// SIMATIC STEP 7 (V5.x) project Desbobinador y cizallado
// CPU: CPU 312
// station: Hardware
// station: SIMATIC 300(1)
// station: P_ADR_BUS

SYMBOL_TABLE
"CONTADOR"	C 1	COUNTER	// Cuenta el numero de planchas cortadas
"Global"	DB 1	DB 1
"Modo1"	DB 2	DB 2
"Modo2"	DB 3	DB 3
"INFO_BOB"	DB 4	DB 4
"DESBOBINADO"	FB 1	FB 1	// Función que se encarga del desbobinado
"CIZALLADO"	FB 2	FB 2	// Funcion que se encaga del cizallado de planchas
"MULT_DESBOB"	FB 3	FB 3
"MULT_CIZA"	FB 4	FB 4
"MULT_GEN"	FB 5	FB 5
"CORTAR"	FC 1	FC 1	// Funcion de cortar las planchas
"PESAJE"	FC 2	FC 2	// Función de pesaje
"MODOS"	FC 3	FC 3	// Gestión de modos
"SCALE"	FC 105	FC 105	// Scaling Values
"PRESENCIA"	I 124.0	BOOL	// Sensor que indica si la bobina está siendo correctamente desbobinada
"SENSOR SARTEN"	I 124.1	BOOL	// Sensor que indica que la plancha ha llegado a la longitud de corte adecuada
"SENSOR CACEROLA"	I 124.2	BOOL	// Sensor que indica que la plancha ha llegado a la longitud de corte adecuada
"SENSOR WOK"	I 124.3	BOOL	// Sensor que indica que la plancha ha llegado a la longitud de corte adecuada
"SENSOR PAELLERA"	I 124.4	BOOL	// Sensor que indica que la plancha ha llegado a la longitud de corte adecuada
"BOBINA COLOCADA"	I 124.5	BOOL	// Sensor que detecta si una bobina ha sido puesta en su lugar para empezar proceso
"SENSOR ABAJO"	I 124.6	BOOL	// Sensor que detecta que la cuchilla de cizallado está abajo
"SENSOR ARRIBA"	I 124.7	BOOL	// Sensor que detecta que la cuchilla de cizallado está arriba
"EXPULSADA"	I 125.0	BOOL	// Sensor que detecta que la plancha recien cortada es expulsada
"MODO A"	I 125.1	BOOL	// Funcionamiento en modo A
"MODO B"	I 125.2	BOOL	// Funcionamiento en modo B
"PALET"	I 125.3	BOOL
"PON"	I 125.4	BOOL
"POFF"	I 125.5	BOOL
"BIT_DE_TRABAJO"	I 125.6	BOOL
"SARTEN"	M 100.1	BOOL	// Peso que corresponde a la bobina para hacer sartenes
"CACEROLA"	M 100.2	BOOL	// Peso que corresponde a la bobina para hacer cacerolas
"WOK"	M 100.3	BOOL	// Peso que corresponde a la bobina para hacer woks
"PAELLERA"	M 100.4	BOOL	// Peso que corresponde a la bobina para hacer paelleras
"CORTADO"	M 100.5	BOOL	// Indica que una plancha ha sido cortada
"X0"	M 101.0	BOOL
"X1"	M 101.1	BOOL
"X2"	M 101.2	BOOL
"X3"	M 101.3	BOOL
"X4"	M 101.4	BOOL
"X5"	M 101.5	BOOL
"X6"	M 101.6	BOOL
"X7"	M 101.7	BOOL
"X8"	M 102.0	BOOL
"X10"	M 102.2	BOOL
"X11"	M 102.3	BOOL
"X20"	M 103.4	BOOL
"X21"	M 103.5	BOOL
"X22"	M 103.6	BOOL
"X23"	M 103.7	BOOL
"X24"	M 104.0	BOOL
"X25"	M 104.1	BOOL
"X30"	M 104.2	BOOL
"X60"	M 104.3	BOOL
"X61"	M 104.4	BOOL
"X62"	M 104.5	BOOL
"X31"	M 104.6	BOOL
"X32"	M 104.7	BOOL
"X33"	M 105.0	BOOL
"X34"	M 105.1	BOOL
"X35"	M 105.2	BOOL
"X40"	M 105.7	BOOL
"X41"	M 106.0	BOOL
"X42"	M 106.1	BOOL
"X43"	M 106.2	BOOL
"X44"	M 106.3	BOOL
"X50"	M 106.7	BOOL
"X51"	M 107.0	BOOL
"X52"	M 107.1	BOOL
"X100"	M 107.2	BOOL
"X101"	M 107.3	BOOL
"X110"	M 107.4	BOOL
"X111"	M 107.5	BOOL
"X53"	M 107.6	BOOL
"X120"	M 107.7	BOOL
"ENDCOUNT"	M 108.0	BOOL	// Marca que avisa del final de la cuenta
"X123"	M 108.2	BOOL
"X124"	M 108.3	BOOL
"X122"	M 108.4	BOOL
"X121"	M 108.5	BOOL
"X54"	M 108.6	BOOL
"STBYDESBOB"	M 108.7	BOOL	// Indica el estado stby del FB1 (desbobinado)
"INIDESBOB"	M 109.0	BOOL	// FP para iniciar el FB1
"INICIZA"	M 109.1	BOOL	// FP para iniciar el FB2
"PLANCHAS"	MW 3	INT	// Numero de planchas por bobina
"OB1"	OB 1	OB 1	// Main programa
"OB100"	OB 100	OB 100	// Inicio del programa
"PESO"	PIW 751	INT	// Sensor de peso que pesa las bobinas
"CENTRO"	PIW 761	INT	// Medida actual del centro
"C_CACEROLA"	PIW 771	INT
"C_SARTEN"	PIW 773	INT
"C_WOK"	PIW 775	INT
"C_PAELLERA"	PIW 777	INT
"ABRIR MCENTRO"	Q 124.1	BOOL	// Salida que hace más grande el centro de sujeción de la bobina
"CERRAR MCENTRO"	Q 124.2	BOOL	// Salida que hace más pequeño el centro de sujeción de la bobina
"DESBOBINAR"	Q 124.3	BOOL	// Actuador que activa la rotación del centro
"EXPULSAR BOBINA"	Q 124.4	BOOL	// Actuador que expulsa el centro de la bobina una vez ha acabado de desbobinar
"BAJAR CUCHILLA"	Q 124.5	BOOL	// Baja la cuchilla, si está a 0 la cuchilla sube
"EXPULSAR PALET"	Q 124.6	BOOL	// Activa un piston que expulsa la plancgha de la zona de corte
"PRENSA"	Q 124.7	BOOL	// Activa la prensa
END_SYMBOL_TABLE

FUNCTION_BLOCK "DESBOBINADO"	// FB 1
TITLE = DESBOBINADO
VERSION : 0.1
VAR_INPUT
  SENSOR : BOOL ;
  PRESENCIA : BOOL ;
  CENTRO : INT ;
  bit_de_trabajo : BOOL ;
  MCENTRO : INT ;
  Contador : COUNTER ;
  START : BOOL ;
  PLANCHAS : WORD  := W#16#100;
END_VAR
VAR_OUTPUT
  ABRIRMCENTRO : BOOL ;
  DESBOBINAR : BOOL ;
  STBY : BOOL ;
END_VAR
VAR
  x31 : BOOL ;
  x32 : BOOL ;
  x33 : BOOL ;
  x34 : BOOL ;
  s1 : BOOL ;
  FP_Bit_Tr : BOOL ;
  x30 : BOOL ;
  FP_PRESENCIA : BOOL ;
  FP_BDT : BOOL ;
  FP_START : BOOL ;
END_VAR
VAR_TEMP
  watchdog_master : BOOL ;
END_VAR
BEGIN
NETWORK
TITLE = Arranque
      SET;
      A     #bit_de_trabajo;
      FP    #FP_BDT;
      S     #x30;
      R     #x31;
      R     #x32;
      R     #x33;
      R     #x34;
      R     #s1;
NETWORK
TITLE = x31 a x32
//Comparacion medida centro con medida nominal del centro para pasar de x31 a x32
      A     #x31;
      A(;
      L     #CENTRO;
      L     #MCENTRO;
      ==R;
      );
      R     #x31;
      S     #x32;
NETWORK
TITLE = x32 a x33
//Presencia detecta que la plancha esta en posicion para empezar el proceso de 
//desbobinado-cizallado
      A     #x32;
      A     #PRESENCIA;
      FP    #FP_PRESENCIA;
      R     #x32;
      S     #x33;
NETWORK
TITLE = x33 a x34
//Detecta que la plancha esta lista para ser cizallada
      A     #x33;
      A     #SENSOR;
      R     #x33;
      S     #x34;
NETWORK
TITLE = x34 a x33
//si el contador no ha acabado
      A     #x34;
      T     LD 1;
      TAK;
      T     LD 5;
      L     #Contador;
      T     LW 9;
      L     LD 5;
      L     LD 1;
      A     C [LW 9];
      AN    #SENSOR;
      R     #x34;
      S     #x33;
NETWORK
TITLE = x34 a s1
//si el contador ha cabado
      A     #x34;
      T     LD 1;
      TAK;
      T     LD 5;
      L     #Contador;
      T     LW 9;
      L     LD 5;
      L     LD 1;
      AN    C [LW 9];
      AN    #SENSOR;
      AN    #PRESENCIA;
      R     #x34;
      S     #x30;
NETWORK
TITLE = Tratamiento de bit de fin
      A     #x30;
      =     #STBY;
NETWORK
TITLE = Abrir centro
      A     #x31;
      =     #ABRIRMCENTRO;
NETWORK
TITLE = Carga del contador y desbobinado en x32
      A     #x32;
      S     #DESBOBINAR;
      L     #PLANCHAS;
      T     LD 1;
      TAK;
      T     LD 5;
      L     #Contador;
      T     LW 9;
      L     LD 5;
      L     LD 1;
      S     C [LW 9];
NETWORK
TITLE = Resta del contador y salida del x33
      A     #x33;
      S     #DESBOBINAR;
NETWORK
TITLE =
      A     #x34;
      R     #DESBOBINAR;
NETWORK
TITLE = De X30 a X31
      A     #x30;
      A     #START;
      FP    #FP_START;
      R     #x30;
      S     #x31;
END_FUNCTION_BLOCK

FUNCTION_BLOCK "CIZALLADO"	// FB 2
TITLE = CIZALLADO
VERSION : 0.1
VAR_INPUT
  bit_de_trabajo : BOOL ;
  SENSOR : BOOL ;
  PLANCHAS : INT ;
  SENSORABAJO : BOOL ;
  SENSORARRIBA : BOOL ;
  EXPULSADA : BOOL ;
  CONTADOR : COUNTER ;
  START : BOOL ;
  STOP : BOOL ;
END_VAR
VAR_OUTPUT
  BAJARCUCHILLA : BOOL ;
  EXPULSARPLANCHA : BOOL ;
  bit_ok : BOOL ;
  bit_error : BOOL ;
  STBY : BOOL ;
END_VAR
VAR
  INICORTAR : BOOL ;
  CORTADO : BOOL ;
  X41 : BOOL ;
  M3 : BOOL ;
  X43 : BOOL ;
  S2 : BOOL ;
  MARCHA : BOOL ;
  PARO : BOOL ;
END_VAR
BEGIN
NETWORK
TITLE = Arranque
      SET;
      FP    #bit_de_trabajo;
      S     #X41;
      R     #M3;
      R     #X43;
      R     #INICORTAR;
      R     #CORTADO;
      R     #bit_ok;
      R     #bit_error;
      R     #S2;
NETWORK
TITLE = De x41 a M3
      A     #X41;
      A     #SENSOR;
      A     #MARCHA;
      R     #X41;
      S     #M3;
NETWORK
TITLE = De M3 a x43
      A     #M3;
      A     #CORTADO;
      R     #M3;
      S     #X43;
NETWORK
TITLE = de x43 a x41
      A     #X43;
      T     LD 0;
      TAK;
      T     LD 4;
      L     #CONTADOR;
      T     LW 8;
      L     LD 4;
      L     LD 0;
      AN    C [LW 8];
      R     #X43;
      S     #X41;
NETWORK
TITLE = de x43 a s2
      A     #X43;
      T     LD 0;
      TAK;
      T     LD 4;
      L     #CONTADOR;
      T     LW 8;
      L     LD 4;
      L     LD 0;
      A     C [LW 8];
      R     #X43;
      S     #S2;
NETWORK
TITLE = De M3 a x43 con call M3
      A     #M3;
      JCN   _001;
      CALL  "CORTAR" (
           bit_de_trabajo           := #INICORTAR,
           SENSORABAJO              := #SENSORABAJO,
           SENSORARRIBA             := #SENSORARRIBA,
           EXPULSADA                := #EXPULSADA,
           BAJARCUCHILLA            := #BAJARCUCHILLA,
           EXPULSARPLANCHA          := #EXPULSARPLANCHA,
           bit_ok                   := #CORTADO);
_001: NOP   0;
      A     #CORTADO;
      R     #M3;
      S     #X43;
NETWORK
TITLE =
      A     #M3;
      =     #INICORTAR;
NETWORK
TITLE = Cuenta el numero de planchas cortadas
      A     #X43;
      T     LD 0;
      TAK;
      T     LD 4;
      L     #CONTADOR;
      T     LW 8;
      L     LD 4;
      L     LD 0;
      CU    C [LW 8];
NETWORK
TITLE =
      A     #MARCHA;
      A     #STOP;
      R     #MARCHA;
      S     #PARO;
NETWORK
TITLE =
      A     #PARO;
      A     #START;
      AN    #STOP;
      R     #PARO;
      S     #MARCHA;
NETWORK
TITLE =
      A     #S2;
      =     #bit_ok;
END_FUNCTION_BLOCK

FUNCTION_BLOCK "MULT_DESBOB"	// FB 3
VERSION : 0.1
VAR_INPUT
  S_CACEROLA : BOOL ;
  S_SARTEN : BOOL ;
  S_WOK : BOOL ;
  S_PAELLERA : BOOL ;
  PRESENCIA : BOOL ;
  C_CACEROLA : INT ;
  C_SARTEN : INT ;
  C_WOK : INT ;
  C_PAELLERA : INT ;
  BIT_DE_TRABAJO : BOOL ;
  MCENTRO : INT ;
  CONTADOR : COUNTER ;
  START : BOOL ;
  STOP : BOOL ;
  PLANCHAS : WORD ;
  SARTEN : BOOL ;
  CACEROLA : BOOL ;
  WOK : BOOL ;
  PAELLERA : BOOL ;
END_VAR
VAR_OUTPUT
  ABRIRMCENTRO : BOOL ;
  DESBOBINAR : BOOL ;
  BIT_OK : BOOL ;
  BIT_ERROR : BOOL ;
  STBY : BOOL ;
END_VAR
VAR
  CAC_DESB : FB 1;
  SART_DESB : FB 1;
  WOK_DESB : FB 1;
  PAELL_DESB : FB 1;
END_VAR
BEGIN
NETWORK
TITLE =
      A     #SARTEN;
      BLD   14;
      =     L 6.0;
      L     DINO;
      T     LW 4;
      CDB;
      OPN   DI [LW 4];
      TAR2  LD 0;
      A     DBX [AR2,P#0.1];
      =     #SART_DESB.SENSOR;
      A     DBX [AR2,P#0.4];
      =     #SART_DESB.PRESENCIA;
      L     DBW [AR2,P#4.0];
      T     #SART_DESB.CENTRO;
      A     DBX [AR2,P#10.0];
      =     #SART_DESB.bit_de_trabajo;
      L     DBW [AR2,P#12.0];
      T     #SART_DESB.MCENTRO;
      L     DBW [AR2,P#14.0];
      T     #SART_DESB.Contador;
      A     DBX [AR2,P#16.0];
      =     #SART_DESB.START;
      A     DBX [AR2,P#16.1];
      =     DIX [AR2,P#52.1];
      L     DBW [AR2,P#18.0];
      T     #SART_DESB.PLANCHAS;
      +AR2  P#42.0;
      UC    "DESBOBINADO";
      LAR2  LD 0;
      A     #SART_DESB.ABRIRMCENTRO;
      =     DBX [AR2,P#22.0];
      A     #SART_DESB.DESBOBINAR;
      =     DBX [AR2,P#22.1];
      A     #SART_DESB.STBY;
      =     DBX [AR2,P#22.2];
      A     DIX [AR2,P#56.3];
      =     DBX [AR2,P#22.3];
      A     DIX [AR2,P#56.4];
      =     DBX [AR2,P#22.4];
      CDB;
      BLD   15;
NETWORK
TITLE =
      A     #CACEROLA;
      BLD   14;
      =     L 6.0;
      L     DINO;
      T     LW 4;
      CDB;
      OPN   DI [LW 4];
      TAR2  LD 0;
      A     DBX [AR2,P#0.0];
      =     #CAC_DESB.SENSOR;
      A     DBX [AR2,P#0.4];
      =     #CAC_DESB.PRESENCIA;
      L     DBW [AR2,P#2.0];
      T     #CAC_DESB.CENTRO;
      A     DBX [AR2,P#10.0];
      =     #CAC_DESB.bit_de_trabajo;
      L     DBW [AR2,P#12.0];
      T     #CAC_DESB.MCENTRO;
      L     DBW [AR2,P#14.0];
      T     #CAC_DESB.Contador;
      A     DBX [AR2,P#16.0];
      =     #CAC_DESB.START;
      A     DBX [AR2,P#16.1];
      =     DIX [AR2,P#34.1];
      L     DBW [AR2,P#18.0];
      T     #CAC_DESB.PLANCHAS;
      +AR2  P#24.0;
      UC    "DESBOBINADO";
      LAR2  LD 0;
      A     #CAC_DESB.ABRIRMCENTRO;
      =     DBX [AR2,P#22.0];
      A     #CAC_DESB.DESBOBINAR;
      =     DBX [AR2,P#22.1];
      A     #CAC_DESB.STBY;
      =     DBX [AR2,P#22.2];
      A     DIX [AR2,P#38.3];
      =     DBX [AR2,P#22.3];
      A     DIX [AR2,P#38.4];
      =     DBX [AR2,P#22.4];
      CDB;
      BLD   15;
NETWORK
TITLE =
      A     #WOK;
      BLD   14;
      =     L 6.0;
      L     DINO;
      T     LW 4;
      CDB;
      OPN   DI [LW 4];
      TAR2  LD 0;
      A     DBX [AR2,P#0.2];
      =     #WOK_DESB.SENSOR;
      A     DBX [AR2,P#0.4];
      =     #WOK_DESB.PRESENCIA;
      L     DBW [AR2,P#6.0];
      T     #WOK_DESB.CENTRO;
      A     DBX [AR2,P#10.0];
      =     #WOK_DESB.bit_de_trabajo;
      L     DBW [AR2,P#12.0];
      T     #WOK_DESB.MCENTRO;
      L     DBW [AR2,P#14.0];
      T     #WOK_DESB.Contador;
      A     DBX [AR2,P#16.0];
      =     #WOK_DESB.START;
      A     DBX [AR2,P#16.1];
      =     DIX [AR2,P#70.1];
      L     DBW [AR2,P#18.0];
      T     #WOK_DESB.PLANCHAS;
      +AR2  P#60.0;
      UC    "DESBOBINADO";
      LAR2  LD 0;
      A     #WOK_DESB.ABRIRMCENTRO;
      =     DBX [AR2,P#22.0];
      A     #WOK_DESB.DESBOBINAR;
      =     DBX [AR2,P#22.1];
      A     #WOK_DESB.STBY;
      =     DBX [AR2,P#22.2];
      A     DIX [AR2,P#74.3];
      =     DBX [AR2,P#22.3];
      A     DIX [AR2,P#74.4];
      =     DBX [AR2,P#22.4];
      CDB;
      BLD   15;
NETWORK
TITLE =
      A     #PAELLERA;
      BLD   14;
      =     L 6.0;
      L     DINO;
      T     LW 4;
      CDB;
      OPN   DI [LW 4];
      TAR2  LD 0;
      A     DBX [AR2,P#0.3];
      =     #PAELL_DESB.SENSOR;
      A     DBX [AR2,P#0.4];
      =     #PAELL_DESB.PRESENCIA;
      L     DBW [AR2,P#8.0];
      T     #PAELL_DESB.CENTRO;
      A     DBX [AR2,P#10.0];
      =     #PAELL_DESB.bit_de_trabajo;
      L     DBW [AR2,P#12.0];
      T     #PAELL_DESB.MCENTRO;
      L     DBW [AR2,P#14.0];
      T     #PAELL_DESB.Contador;
      A     DBX [AR2,P#16.0];
      =     #PAELL_DESB.START;
      A     DBX [AR2,P#16.1];
      =     DIX [AR2,P#88.1];
      L     DBW [AR2,P#18.0];
      T     #PAELL_DESB.PLANCHAS;
      +AR2  P#78.0;
      UC    "DESBOBINADO";
      LAR2  LD 0;
      A     #PAELL_DESB.ABRIRMCENTRO;
      =     DBX [AR2,P#22.0];
      A     #PAELL_DESB.DESBOBINAR;
      =     DBX [AR2,P#22.1];
      A     #PAELL_DESB.STBY;
      =     DBX [AR2,P#22.2];
      A     DIX [AR2,P#92.3];
      =     DBX [AR2,P#22.3];
      A     DIX [AR2,P#92.4];
      =     DBX [AR2,P#22.4];
      CDB;
      BLD   15;
END_FUNCTION_BLOCK

FUNCTION_BLOCK "MULT_CIZA"	// FB 4
VERSION : 0.1
VAR_INPUT
  S_CACEROLA : BOOL ;
  S_WOK : BOOL ;
  S_SARTEN : BOOL ;
  S_PAELLERA : BOOL ;
  BIT_DE_TRABAJO : BOOL ;
  PLANCHAS : INT ;
  SENSORARRIBA : BOOL ;
  SENSORABAJO : BOOL ;
  EXPULSADA : BOOL ;
  CONTADOR : COUNTER ;
  SARTEN : BOOL ;
  CACEROLA : BOOL ;
  WOK : BOOL ;
  PAELLERA : BOOL ;
  START : BOOL ;
  STOP : BOOL ;
END_VAR
VAR_OUTPUT
  EXPULSARPLANCHA : BOOL ;
  BAJARCUCHILLA : BOOL ;
  BIT_OK : BOOL ;
END_VAR
VAR
  CAC_CIZA : FB 2;
  SART_CIZA : FB 2;
  WOK_CIZA : FB 2;
  PAELL_CIZA : FB 2;
  STBY : BOOL ;
END_VAR
BEGIN
NETWORK
TITLE =
      A     #CACEROLA;
      BLD   14;
      =     L 6.0;
      L     DINO;
      T     LW 4;
      CDB;
      OPN   DI [LW 4];
      TAR2  LD 0;
      A     DBX [AR2,P#0.4];
      =     #CAC_CIZA.bit_de_trabajo;
      A     DBX [AR2,P#0.0];
      =     #CAC_CIZA.SENSOR;
      L     DBW [AR2,P#2.0];
      T     #CAC_CIZA.PLANCHAS;
      A     DBX [AR2,P#4.1];
      =     #CAC_CIZA.SENSORABAJO;
      A     DBX [AR2,P#4.0];
      =     #CAC_CIZA.SENSORARRIBA;
      A     DBX [AR2,P#4.2];
      =     #CAC_CIZA.EXPULSADA;
      L     DBW [AR2,P#6.0];
      T     #CAC_CIZA.CONTADOR;
      A     DBX [AR2,P#8.4];
      =     #CAC_CIZA.START;
      A     DBX [AR2,P#8.5];
      =     #CAC_CIZA.STOP;
      +AR2  P#12.0;
      UC    "CIZALLADO";
      LAR2  LD 0;
      A     #CAC_CIZA.BAJARCUCHILLA;
      =     DBX [AR2,P#10.1];
      A     #CAC_CIZA.EXPULSARPLANCHA;
      =     DBX [AR2,P#10.0];
      A     #CAC_CIZA.bit_ok;
      =     DBX [AR2,P#10.2];
      A     #CAC_CIZA.STBY;
      =     DBX [AR2,P#68.0];
      CDB;
      BLD   15;
NETWORK
TITLE =
      A     #WOK;
      BLD   14;
      =     L 6.0;
      L     DINO;
      T     LW 4;
      CDB;
      OPN   DI [LW 4];
      TAR2  LD 0;
      A     DBX [AR2,P#0.4];
      =     #WOK_CIZA.bit_de_trabajo;
      A     DBX [AR2,P#0.1];
      =     #WOK_CIZA.SENSOR;
      L     DBW [AR2,P#2.0];
      T     #WOK_CIZA.PLANCHAS;
      A     DBX [AR2,P#4.1];
      =     #WOK_CIZA.SENSORABAJO;
      A     DBX [AR2,P#4.0];
      =     #WOK_CIZA.SENSORARRIBA;
      A     DBX [AR2,P#4.2];
      =     #WOK_CIZA.EXPULSADA;
      L     DBW [AR2,P#6.0];
      T     #WOK_CIZA.CONTADOR;
      A     DBX [AR2,P#8.4];
      =     #WOK_CIZA.START;
      A     DBX [AR2,P#8.5];
      =     #WOK_CIZA.STOP;
      +AR2  P#40.0;
      UC    "CIZALLADO";
      LAR2  LD 0;
      A     #WOK_CIZA.BAJARCUCHILLA;
      =     DBX [AR2,P#10.1];
      A     #WOK_CIZA.EXPULSARPLANCHA;
      =     DBX [AR2,P#10.0];
      A     #WOK_CIZA.bit_ok;
      =     DBX [AR2,P#10.2];
      A     #WOK_CIZA.STBY;
      =     DBX [AR2,P#68.0];
      CDB;
      BLD   15;
NETWORK
TITLE =
      A     #SARTEN;
      BLD   14;
      =     L 6.0;
      L     DINO;
      T     LW 4;
      CDB;
      OPN   DI [LW 4];
      TAR2  LD 0;
      A     DBX [AR2,P#0.4];
      =     #SART_CIZA.bit_de_trabajo;
      A     DBX [AR2,P#0.2];
      =     #SART_CIZA.SENSOR;
      L     DBW [AR2,P#2.0];
      T     #SART_CIZA.PLANCHAS;
      A     DBX [AR2,P#4.1];
      =     #SART_CIZA.SENSORABAJO;
      A     DBX [AR2,P#4.0];
      =     #SART_CIZA.SENSORARRIBA;
      A     DBX [AR2,P#4.2];
      =     #SART_CIZA.EXPULSADA;
      L     DBW [AR2,P#6.0];
      T     #SART_CIZA.CONTADOR;
      A     DBX [AR2,P#8.4];
      =     #SART_CIZA.START;
      A     DBX [AR2,P#8.5];
      =     #SART_CIZA.STOP;
      +AR2  P#26.0;
      UC    "CIZALLADO";
      LAR2  LD 0;
      A     #SART_CIZA.BAJARCUCHILLA;
      =     DBX [AR2,P#10.1];
      A     #SART_CIZA.EXPULSARPLANCHA;
      =     DBX [AR2,P#10.0];
      A     #SART_CIZA.bit_ok;
      =     DBX [AR2,P#10.2];
      A     #SART_CIZA.STBY;
      =     DBX [AR2,P#68.0];
      CDB;
      BLD   15;
NETWORK
TITLE =
      A     #PAELLERA;
      BLD   14;
      =     L 6.0;
      L     DINO;
      T     LW 4;
      CDB;
      OPN   DI [LW 4];
      TAR2  LD 0;
      A     DBX [AR2,P#0.4];
      =     #PAELL_CIZA.bit_de_trabajo;
      A     DBX [AR2,P#0.3];
      =     #PAELL_CIZA.SENSOR;
      L     DBW [AR2,P#2.0];
      T     #PAELL_CIZA.PLANCHAS;
      A     DBX [AR2,P#4.1];
      =     #PAELL_CIZA.SENSORABAJO;
      A     DBX [AR2,P#4.0];
      =     #PAELL_CIZA.SENSORARRIBA;
      A     DBX [AR2,P#4.2];
      =     #PAELL_CIZA.EXPULSADA;
      L     DBW [AR2,P#6.0];
      T     #PAELL_CIZA.CONTADOR;
      A     DBX [AR2,P#8.4];
      =     #PAELL_CIZA.START;
      A     DBX [AR2,P#8.5];
      =     #PAELL_CIZA.STOP;
      +AR2  P#54.0;
      UC    "CIZALLADO";
      LAR2  LD 0;
      A     #PAELL_CIZA.BAJARCUCHILLA;
      =     DBX [AR2,P#10.1];
      A     #PAELL_CIZA.EXPULSARPLANCHA;
      =     DBX [AR2,P#10.0];
      A     #PAELL_CIZA.bit_ok;
      =     DBX [AR2,P#10.2];
      A     #PAELL_CIZA.STBY;
      =     DBX [AR2,P#68.0];
      CDB;
      BLD   15;
END_FUNCTION_BLOCK

FUNCTION_BLOCK "MULT_GEN"	// FB 5
VERSION : 0.1
VAR_INPUT
  MODO : BOOL ;
  BIT_DE_TRABAJO : BOOL ;
  START : BOOL ;
  STOP : BOOL ;
  BOBINA_COLOCADA : BOOL ;
  IN_SCALE : INT ;
  S_CACEROLA : BOOL ;
  S_WOK : BOOL ;
  S_PAELLERA : BOOL ;
  S_SARTEN : BOOL ;
  PRESENCIA : BOOL ;
  MCENTRO : INT ;
  CONTADOR : COUNTER ;
END_VAR
VAR_OUTPUT
  ABRIRMCENTRO : BOOL ;
END_VAR
VAR_IN_OUT
  DESBOBINAR : BOOL ;
END_VAR
VAR
  CIZALLADO : FB 4;
  DESBOBINADO : FB 3;
  X0 : BOOL ;
  MARCHA : BOOL ;
  PARO : BOOL ;
  X1 : BOOL ;
  M4 : BOOL ;
  M1 : BOOL ;
  X7 : BOOL ;
  X8 : BOOL ;
  X10 : BOOL ;
  X11 : BOOL ;
  X20 : BOOL ;
  M2 : BOOL ;
  X25 : BOOL ;
  OK_SCALE : BOOL ;
  START_SCALE : BOOL ;
  STOP_SCALE : BOOL ;
  STBY_SCALE : BOOL ;
  SARTEN : BOOL ;
  CACEROLA : BOOL ;
  WOK : BOOL ;
  PAELLERA : BOOL ;
  START_DESBOBINADO : BOOL ;
  STOP_DESBOBINADO : BOOL ;
END_VAR
BEGIN
NETWORK
TITLE =
      A     #BIT_DE_TRABAJO;
      S     #X0;
      S     #PARO;
      R     #MARCHA;
      R     #X1;
      R     #M4;
      R     #M1;
      R     #X7;
      R     #X8;
      R     #X10;
      R     #X11;
      R     #X20;
      R     #M2;
      R     #X25;
NETWORK
TITLE =
      A     #MARCHA;
      A     #STOP;
      R     #MARCHA;
      S     #PARO;
NETWORK
TITLE =
      A     #PARO;
      A     #START;
      AN    #STOP;
      R     #PARO;
      S     #MARCHA;
NETWORK
TITLE =
      A     #X0;
      A     #MARCHA;
      R     #X0;
      S     #X1;
      S     #X10;
      S     #X20;
NETWORK
TITLE =
      A     #X1;
      A     #BOBINA_COLOCADA;
      R     #X1;
      S     #M4;
NETWORK
TITLE =
      A     #M4;
      JCN   _001;
      CALL  "PESAJE" (
           in                       := #IN_SCALE,
           PESO_SARTEN              := "Global".PESO_SARTEN,
           PESO_CACEROLA            := "Global".PESO_CACEROLA,
           PESO_WOK                 := "Global".PESO_WOK,
           PESO_PAELLERA            := "Global".PESO_PAELLERA,
           bit_de_trabajo           := #BIT_DE_TRABAJO,
           RECIBIDO                 := #OK_SCALE,
           START                    := #START_SCALE,
           STOP                     := #STOP_SCALE,
           stby                     := #STBY_SCALE,
           SARTEN                   := #SARTEN,
           CACEROLA                 := #CACEROLA,
           WOK                      := #WOK,
           PAELLERA                 := #PAELLERA);
_001: NOP   0;
NETWORK
TITLE =
      A     #M4;
      =     #START_SCALE;
NETWORK
TITLE =
      A     #M4;
      A(;
      A     #SARTEN;
      O     #WOK;
      O     #PAELLERA;
      O     #CACEROLA;
      );
      JCN   _002;
      BLD   14;
      =     L 6.0;
      L     DINO;
      T     LW 4;
      CDB;
      OPN   DI [LW 4];
      TAR2  LD 0;
      A     DBX [AR2,P#4.0];
      =     #DESBOBINADO.S_CACEROLA;
      A     DBX [AR2,P#4.3];
      =     #DESBOBINADO.S_SARTEN;
      A     DBX [AR2,P#4.1];
      =     #DESBOBINADO.S_WOK;
      A     DBX [AR2,P#4.2];
      =     #DESBOBINADO.S_PAELLERA;
      A     DBX [AR2,P#4.4];
      =     #DESBOBINADO.PRESENCIA;
      OPN   DI 4;
      L     DIW 0;
      OPN   DI [LW 4];
      T     #DESBOBINADO.C_CACEROLA;
      OPN   DI 4;
      L     DIW 2;
      OPN   DI [LW 4];
      T     #DESBOBINADO.C_SARTEN;
      OPN   DI 4;
      L     DIW 4;
      OPN   DI [LW 4];
      T     #DESBOBINADO.C_WOK;
      OPN   DI 4;
      L     DIW 6;
      OPN   DI [LW 4];
      T     #DESBOBINADO.C_PAELLERA;
      A     DBX [AR2,P#0.1];
      =     #DESBOBINADO.BIT_DE_TRABAJO;
      L     DBW [AR2,P#6.0];
      T     #DESBOBINADO.MCENTRO;
      L     DBW [AR2,P#8.0];
      T     #DESBOBINADO.CONTADOR;
      A     DBX [AR2,P#182.5];
      =     #DESBOBINADO.START;
      A     DBX [AR2,P#182.6];
      =     #DESBOBINADO.STOP;
      OPN   DI 1;
      L     DIW 16;
      OPN   DI [LW 4];
      T     #DESBOBINADO.PLANCHAS;
      A     DBX [AR2,P#182.1];
      =     #DESBOBINADO.SARTEN;
      A     DBX [AR2,P#182.2];
      =     #DESBOBINADO.CACEROLA;
      A     DBX [AR2,P#182.3];
      =     #DESBOBINADO.WOK;
      A     DBX [AR2,P#182.4];
      =     #DESBOBINADO.PAELLERA;
      +AR2  P#84.0;
      UC    "MULT_DESBOB";
      LAR2  LD 0;
      A     #DESBOBINADO.ABRIRMCENTRO;
      =     DBX [AR2,P#10.0];
      A     #DESBOBINADO.DESBOBINAR;
      =     DBX [AR2,P#12.0];
      CDB;
      BLD   15;
_002: NOP   0;
END_FUNCTION_BLOCK

FUNCTION "CORTAR" : VOID	// FC 1
TITLE = CORTAR
VERSION : 0.1
VAR_INPUT
  bit_de_trabajo : BOOL ;
  SENSORABAJO : BOOL ;
  SENSORARRIBA : BOOL ;
  EXPULSADA : BOOL ;
END_VAR
VAR_OUTPUT
  BAJARCUCHILLA : BOOL ;
  EXPULSARPLANCHA : BOOL ;
  bit_ok : BOOL ;
END_VAR
VAR_TEMP
  x51 : BOOL ;
  x52 : BOOL ;
  x53 : BOOL ;
  s3 : BOOL ;
END_VAR
BEGIN
NETWORK
TITLE = Arranque
      SET;
      FP    #bit_de_trabajo;
      S     #x51;
      R     #x52;
      R     #x53;
      R     #s3;
NETWORK
TITLE = de x51 a x52
      A     #x51;
      A     #SENSORABAJO;
      R     #x51;
      S     #x52;
NETWORK
TITLE = de x52 a x53
      A     #x52;
      A     #SENSORARRIBA;
      R     #x52;
      S     #x53;
NETWORK
TITLE = de x53 a s3
      A     #x53;
      A     #EXPULSADA;
      R     #x53;
      S     #s3;
NETWORK
TITLE = Accion x51
      A     "X51";
      =     #BAJARCUCHILLA;
NETWORK
TITLE = Accion x53
      A     #x53;
      =     #EXPULSARPLANCHA;
NETWORK
TITLE = Accion final
      A     #s3;
      =     #bit_ok;
END_FUNCTION

FUNCTION "PESAJE" : VOID	// FC 2
TITLE = PESAJE
VERSION : 0.1
VAR_INPUT
  in : INT ;
  PESO_SARTEN : REAL ;
  PESO_CACEROLA : REAL ;
  PESO_WOK : REAL ;
  PESO_PAELLERA : REAL ;
  bit_de_trabajo : BOOL ;
  RECIBIDO : BOOL ;
  START : BOOL ;
  STOP : BOOL ;
END_VAR
VAR_OUTPUT
  stby : BOOL ;
  SARTEN : BOOL ;
  CACEROLA : BOOL ;
  WOK : BOOL ;
  PAELLERA : BOOL ;
END_VAR
VAR_TEMP
  retFC105 : WORD ;
  PESO : REAL ;
  x121 : BOOL ;
  x122 : BOOL ;
  x123 : BOOL ;
  x124 : BOOL ;
  m3 : BOOL ;
  x120 : BOOL ;
  MARCHA : BOOL ;
  PARO : BOOL ;
END_VAR
BEGIN
NETWORK
TITLE = Pesado
      A     #m3;
      CALL  "SCALE" (
           $1                       := #in,
           $2                       := L#1133903872,
           $3                       := L#0,
           $4                       := FALSE,
           $5                       := #retFC105,
           $6                       := #PESO);
NETWORK
TITLE = Arranque
      SET;
      FP    #bit_de_trabajo;
      S     #m3;
      R     #x121;
      R     #x122;
      R     #x123;
      R     #x124;
NETWORK
TITLE = COMPARACION PESO CON PESO_SARTEN
      A(;
      L     #PESO;
      A(;
      L     #PESO_SARTEN;
      L     5.000000e+00;
      +R;
      );
      <=R;
      );
      A(;
      L     #PESO;
      A(;
      L     #PESO_SARTEN;
      L     5.000000e+00;
      -R;
      );
      >=R;
      );
      A     #MARCHA;
      S     #x121;
      R     #m3;
NETWORK
TITLE = COMPARACION PESO CON PESO_CACEROLA
      A(;
      L     #PESO;
      A(;
      L     #PESO_CACEROLA;
      L     5.000000e+00;
      +R;
      );
      <=R;
      );
      A(;
      L     #PESO;
      A(;
      L     #PESO_CACEROLA;
      L     5.000000e+00;
      -R;
      );
      >=R;
      );
      A     #MARCHA;
      S     #x122;
      R     #m3;
NETWORK
TITLE = COMPARACION PESO PESO_WOK
      A(;
      L     #PESO;
      A(;
      L     #PESO_WOK;
      L     5.000000e+00;
      +R;
      );
      <=R;
      );
      A(;
      L     #PESO;
      A(;
      L     #PESO_WOK;
      L     5.000000e+00;
      -R;
      );
      >=R;
      );
      A     #MARCHA;
      S     #x123;
      R     #m3;
NETWORK
TITLE = COMPARACION PESO CON PESO_PAELLERA
      A(;
      L     #PESO;
      A(;
      L     #PESO_PAELLERA;
      L     5.000000e+00;
      +R;
      );
      <=R;
      );
      A(;
      L     #PESO;
      A(;
      L     #PESO_PAELLERA;
      L     5.000000e+00;
      -R;
      );
      >=R;
      );
      A     #MARCHA;
      S     #x124;
      R     #m3;
NETWORK
TITLE = TRATAMIENTO SALIDAS
      A     #x121;
      =     #SARTEN;
      A     #x122;
      =     #CACEROLA;
      A     #x123;
      =     #WOK;
      A     #x124;
      =     #PAELLERA;
NETWORK
TITLE = Paso de estado pesado a stby
      A(;
      A     #x121;
      O     #x122;
      O     #x123;
      O     #x124;
      );
      A     #RECIBIDO;
      R     #x121;
      R     #x122;
      R     #x123;
      R     #x124;
      S     #x120;
NETWORK
TITLE = Salida STBY
      A     #x120;
      =     #stby;
NETWORK
TITLE = MARCHA PARO
      A     #MARCHA;
      A     #STOP;
      R     #MARCHA;
      S     #PARO;
NETWORK
TITLE = PARO MARCHA
      A     #PARO;
      A     #START;
      AN    #STOP;
      R     #PARO;
      S     #MARCHA;
END_FUNCTION

FUNCTION "MODOS" : VOID	// FC 3
TITLE = GESTION DE MODOS
VERSION : 0.1
VAR_INPUT
  MODO1 : BOOL ;
  MODO2 : BOOL ;
END_VAR
VAR_OUTPUT
  CONTADOR : INT ;
  PSARTEN : INT ;
  PCACEROLA : INT ;
  PWOK : INT ;
  PPAELLERA : INT ;
END_VAR
VAR_TEMP
  X60 : BOOL ;
  X61 : BOOL ;
  X62 : BOOL ;
END_VAR
BEGIN
NETWORK
TITLE = De X60 a X61
      A     #X60;
      A     #MODO1;
      R     #X60;
      S     #X61;
NETWORK
TITLE = De X61 a X60
      A     #X61;
      AN    #MODO1;
      R     #X61;
      S     #X60;
NETWORK
TITLE = De X60 a X62
      A     #X60;
      A     #MODO2;
      R     #X60;
      S     #X62;
NETWORK
TITLE = De X62 a X60
      A     #X62;
      AN    #MODO2;
      R     #X62;
      S     #X60;
NETWORK
TITLE = Numero de planchas por bobina y peso Modo 1
      A     #X61;
      L     "Modo1".PLANCHAS;
      T     "Global".PLANCHAS;
      L     "Modo1".PESO_PAELLERA;
      T     "Global".PESO_PAELLERA;
      L     "Modo1".PESO_WOK;
      T     "Global".PESO_WOK;
      L     "Modo1".PESO_SARTEN;
      T     "Global".PESO_SARTEN;
      L     "Modo1".PESO_CACEROLA;
      T     "Global".PESO_CACEROLA;
NETWORK
TITLE =
      A     #X62;
      L     "Modo2".PLANCHAS;
      T     "Global".PLANCHAS;
      L     "Modo2".PESO_PAELLERA;
      T     "Global".PESO_PAELLERA;
      L     "Modo2".PESO_WOK;
      T     "Global".PESO_WOK;
      L     "Modo2".PESO_SARTEN;
      T     "Global".PESO_SARTEN;
      L     "Modo2".PESO_CACEROLA;
      T     "Global".PESO_CACEROLA;
NETWORK
TITLE = Numero de planchas por bobina y peso Modo 2
      A     #X62;
      L     #CONTADOR;
      OPN   DB 200;
      L     #PSARTEN;
      OPN   DB 200;
      L     #PCACEROLA;
      OPN   DB 220;
      L     #PWOK;
      OPN   DB 240;
      L     #PPAELLERA;
      OPN   DB 260;
END_FUNCTION

// FC 105: know-how protected block, not included

DATA_BLOCK "Global"	// DB 1
VERSION : 0.1
  STRUCT
   PESO_CACEROLA : REAL ;	//Peso Bobina Cacerolas
   PESO_WOK : REAL ;	//Peso Bobina Wok
   PESO_SARTEN : REAL ;	//Peso Bobina Sarten
   PESO_PAELLERA : REAL ;	//Peso Bobina Paellera
   PLANCHAS : WORD ;	//Número de planchas por bobina
  END_STRUCT ;	
BEGIN
   PESO_CACEROLA := 1.000000e+02;
   PESO_WOK := 1.100000e+02;
   PESO_SARTEN := 1.200000e+02;
   PESO_PAELLERA := 1.300000e+02;
   PLANCHAS := W#16#100;
END_DATA_BLOCK

DATA_BLOCK "Modo1"	// DB 2
VERSION : 0.1
  STRUCT
   PESO_CACEROLA : REAL  := 1.000000e+002;	//Peso Bobina Cacerolas
   PESO_WOK : REAL  := 1.100000e+002;	//Peso Bobina Wok
   PESO_SARTEN : REAL  := 1.200000e+002;	//Peso Bobina Sarten
   PESO_PAELLERA : REAL  := 1.300000e+002;	//Peso Bobina Paellera
   PLANCHAS : WORD  := W#16#100;	//Número de planchas por bobina
  END_STRUCT ;	
BEGIN
   PESO_CACEROLA := 1.000000e+02;
   PESO_WOK := 1.100000e+02;
   PESO_SARTEN := 1.200000e+02;
   PESO_PAELLERA := 1.300000e+02;
   PLANCHAS := W#16#100;
END_DATA_BLOCK

DATA_BLOCK "Modo2"	// DB 3
VERSION : 0.1
  STRUCT
   PESO_CACEROLA : REAL  := 2.000000e+002;	//Peso Bobina Cacerolas
   PESO_WOK : REAL  := 2.200000e+002;	//Peso Bobina Wok
   PESO_SARTEN : REAL  := 2.400000e+002;	//Peso Bobina Sarten
   PESO_PAELLERA : REAL  := 2.600000e+002;	//Peso Bobina Paellera
   PLANCHAS : WORD  := W#16#200;	//Número de planchas por bobina
  END_STRUCT ;	
BEGIN
   PESO_CACEROLA := 2.000000e+02;
   PESO_WOK := 2.200000e+02;
   PESO_SARTEN := 2.400000e+02;
   PESO_PAELLERA := 2.600000e+02;
   PLANCHAS := W#16#200;
END_DATA_BLOCK

DATA_BLOCK "INFO_BOB"	// DB 4
VERSION : 0.1
  STRUCT
   CENTRO_CACEROLA : INT ;	//Variable provisional
   CENTRO_SARTEN : INT ;
   CENTRO_WOK : INT ;
   CENTRO_PAELLERA : INT ;
  END_STRUCT ;	
BEGIN
END_DATA_BLOCK

ORGANIZATION_BLOCK "OB1"	// OB 1
TITLE = "Main Program Sweep (Cycle)"
VERSION : 0.1
VAR_TEMP
  OB1_EV_CLASS : BYTE ;	//Bits 0-3 = 1 (Coming event), Bits 4-7 = 1 (Event class 1)
  OB1_SCAN_1 : BYTE ;	//1 (Cold restart scan 1 of OB 1), 3 (Scan 2-n of OB 1)
  OB1_PRIORITY : BYTE ;	//Priority of OB Execution
  OB1_OB_NUMBR : BYTE ;	//1 (Organization block 1, OB1)
  OB1_RESERVED_1 : BYTE ;	//Reserved for system
  OB1_RESERVED_2 : BYTE ;	//Reserved for system
  OB1_PREV_CYCLE : INT ;	//Cycle time of previous OB1 scan (milliseconds)
  OB1_MIN_CYCLE : INT ;	//Minimum cycle time of OB1 (milliseconds)
  OB1_MAX_CYCLE : INT ;	//Maximum cycle time of OB1 (milliseconds)
  OB1_DATE_TIME : DATE_AND_TIME ;	//Date and time OB1 started
END_VAR
BEGIN
NETWORK
TITLE =
      A     "X100";
      A     "PON";
      AN    "POFF";
      R     "X100";
      S     "X101";
NETWORK
TITLE =
      A     "X101";
      A     "POFF";
      R     "X101";
      S     "X100";
NETWORK
TITLE =
      A     "X0";
      A     "X101";
      AN    "X60";
      R     "X0";
      S     "X1";
      S     "X10";
      S     "X20";
NETWORK
TITLE =
      A     "X1";
      A     "BOBINA COLOCADA";
      R     "X1";
      S     "X2";
NETWORK
TITLE =
      A     "X2";
      A     DB1.DBX 4.1;
      R     "X2";
      S     "X3";
NETWORK
TITLE =
      A     "X2";
      A     DB2.DBX 4.1;
      R     "X2";
      S     "X4";
NETWORK
TITLE =
      A     "X2";
      A     DB3.DBX 4.1;
      R     "X2";
      S     "X5";
NETWORK
TITLE =
      A     "X2";
      A     DB4.DBX 4.1;
      R     "X2";
      S     "X6";
NETWORK
TITLE =
      A     "X3";
      O     "X4";
      O     "X5";
      O     "X6";
      R     "X121";
      R     "X122";
      R     "X123";
      R     "X124";
      S     "X120";
NETWORK
TITLE =
      A(;
      A     "X3";
      O     "X4";
      O     "X5";
      O     "X6";
      );
      A     "X30";
      R     "X3";
      R     "X4";
      R     "X5";
      R     "X6";
      S     "X7";
NETWORK
TITLE =
      A     "X7";
      A(;
      L     PIW 753;
      L     0;
      ==R;
      );
      R     "X7";
      S     "X8";
NETWORK
TITLE =
      A     "X8";
      A     "X101";
      AN    "BOBINA COLOCADA";
      R     "X8";
      S     "X1";
NETWORK
TITLE =
      A     "X10";
      A     "DESBOBINAR";
      A     "X101";
      R     "X10";
      S     "X11";
NETWORK
TITLE =
      A     "X20";
      A     DB1.DBX 4.1;
      R     "X20";
      S     "X21";
NETWORK
TITLE =
      A     "X20";
      A     DB2.DBX 4.1;
      R     "X20";
      S     "X22";
NETWORK
TITLE =
      A     "X20";
      A     DB3.DBX 4.1;
      R     "X20";
      S     "X23";
NETWORK
TITLE =
      A     "X20";
      A     DB4.DBX 4.1;
      R     "X20";
      S     "X24";
      A     "X40";
NETWORK
TITLE =
      A(;
      A     "X21";
      O     "X22";
      O     "X23";
      O     "X24";
      );
      A     "X30";
      R     "X21";
      R     "X22";
      R     "X23";
      R     "X24";
      S     "X25";
NETWORK
TITLE =
      A     "X25";
      A     "X101";
      AN    "PALET";
      R     "X25";
      S     "X20";
NETWORK
TITLE =
      A(;
      A     "X8";
      AN    "BOBINA COLOCADA";
      );
      A     "X10";
      A(;
      A     "X25";
      AN    "PALET";
      );
      A     "X100";
      R     "X8";
      R     "X10";
      R     "X25";
      S     "X0";
NETWORK
TITLE =
      A     "X0";
      CALL  "MODOS" (
           $1                       := "MODO A",
           $2                       := "MODO B",
           $3                       := "PLANCHAS",
           $4                       := DB1.DBW 2,
           $5                       := DB2.DBW 2,
           $6                       := DB3.DBW 2,
           $7                       := "INFO_BOB".CENTRO_SARTEN,
           $8                       := "X60",
           $9                       := "X61",
           $10                      := "X62");
NETWORK
TITLE =
      A     "X2";
      CALL  "PESAJE" (
           $1                       := P#P 752.0,
           $2                       := DB1.DBX 4.1,
           $3                       := DB2.DBX 4.1,
           $4                       := DB3.DBX 4.1,
           $5                       := DB4.DBX 4.1);
NETWORK
TITLE = Salida que hace más pequeño el centro de sujeción de la bobina
      A     "X7";
      S     "CERRAR MCENTRO";
NETWORK
TITLE = Salida que hace más pequeño el centro de sujeción de la bobina
      A     "X8";
      R     "CERRAR MCENTRO";
      S     "EXPULSAR BOBINA";
NETWORK
TITLE = Activa la prensa
      A     "X11";
      S     "PRENSA";
NETWORK
TITLE = Activa la prensa
      A     "X10";
      R     "PRENSA";
NETWORK
TITLE = Activa un piston que expulsa la plancgha de la zona de corte
      A     "X20";
      R     "EXPULSAR PALET";
NETWORK
TITLE = Activa un piston que expulsa la plancgha de la zona de corte
      A     "X25";
      S     "EXPULSAR PALET";
NETWORK
TITLE =
      A     "X2";
      BLD   3;
      =     L 24.0;
      CDB;
      OPN   DI 5;
      TAR2  LD 20;
      OPN   DI 1;
      A     DIX 4.0;
      OPN   DI 5;
      =     DIX 0.0;
      A     "PRESENCIA";
      =     DIX 0.1;
      OPN   DI 1;
      L     DIW 0;
      OPN   DI 5;
      T     DIW 2;
      L     "PLANCHAS";
      T     DIW 4;
      A     "INIDESBOB";
      =     DIX 6.0;
      L     PIW 752;
      T     DIW 8;
      LAR2  P#DBX 0.0;
      UC    "DESBOBINADO";
      LAR2  LD 20;
      A     DIX 10.0;
      =     "ABRIR MCENTRO";
      A     DIX 10.1;
      =     "CERRAR MCENTRO";
      A     DIX 10.2;
      =     "DESBOBINAR";
      A     DIX 10.3;
      =     "STBYDESBOB";
      CDB;
      BLD   4;
      FP    "INIDESBOB";
NETWORK
TITLE =
      A     "X3";
      BLD   3;
      =     L 24.0;
      CDB;
      OPN   DI 5;
      TAR2  LD 20;
      OPN   DI 2;
      A     DIX 4.0;
      OPN   DI 5;
      =     DIX 0.0;
      A     "PRESENCIA";
      =     DIX 0.1;
      OPN   DI 2;
      L     DIW 0;
      OPN   DI 5;
      T     DIW 2;
      L     "PLANCHAS";
      T     DIW 4;
      A     "INIDESBOB";
      =     DIX 6.0;
      L     PIW 752;
      T     DIW 8;
      LAR2  P#DBX 0.0;
      UC    "DESBOBINADO";
      LAR2  LD 20;
      A     DIX 10.0;
      =     "ABRIR MCENTRO";
      A     DIX 10.1;
      =     "CERRAR MCENTRO";
      A     DIX 10.2;
      =     "DESBOBINAR";
      A     DIX 10.3;
      =     "STBYDESBOB";
      CDB;
      BLD   4;
      FP    "INIDESBOB";
NETWORK
TITLE =
      A     "X5";
      BLD   3;
      =     L 24.0;
      CDB;
      OPN   DI 5;
      TAR2  LD 20;
      OPN   DI 3;
      A     DIX 4.0;
      OPN   DI 5;
      =     DIX 0.0;
      A     "PRESENCIA";
      =     DIX 0.1;
      OPN   DI 3;
      L     DIW 0;
      OPN   DI 5;
      T     DIW 2;
      L     "PLANCHAS";
      T     DIW 4;
      A     "INIDESBOB";
      =     DIX 6.0;
      L     PIW 752;
      T     DIW 8;
      LAR2  P#DBX 0.0;
      UC    "DESBOBINADO";
      LAR2  LD 20;
      A     DIX 10.0;
      =     "ABRIR MCENTRO";
      A     DIX 10.1;
      =     "CERRAR MCENTRO";
      A     DIX 10.2;
      =     "DESBOBINAR";
      A     DIX 10.3;
      =     "STBYDESBOB";
      CDB;
      BLD   4;
      FP    "INIDESBOB";
NETWORK
TITLE =
      A     "X6";
      BLD   3;
      =     L 24.0;
      CDB;
      OPN   DI 5;
      TAR2  LD 20;
      OPN   DI 4;
      A     DIX 4.0;
      OPN   DI 5;
      =     DIX 0.0;
      A     "PRESENCIA";
      =     DIX 0.1;
      OPN   DI 4;
      L     DIW 0;
      OPN   DI 5;
      T     DIW 2;
      L     "PLANCHAS";
      T     DIW 4;
      A     "INIDESBOB";
      =     DIX 6.0;
      L     PIW 752;
      T     DIW 8;
      LAR2  P#DBX 0.0;
      UC    "DESBOBINADO";
      LAR2  LD 20;
      A     DIX 10.0;
      =     "ABRIR MCENTRO";
      A     DIX 10.1;
      =     "CERRAR MCENTRO";
      A     DIX 10.2;
      =     "DESBOBINAR";
      A     DIX 10.3;
      =     "STBYDESBOB";
      CDB;
      BLD   4;
      FP    "INIDESBOB";
NETWORK
TITLE =
      A     "X21";
      CALL  "CIZALLADO" , DB 6 (
           bit_de_trabajo           := "INICIZA",
           SENSOR                   := DB1.DBX 4.0,
           PLANCHAS                 := "PLANCHAS");
      FP    "INICIZA";
NETWORK
TITLE =
      A     "X22";
      CALL  "CIZALLADO" , DB 6 (
           bit_de_trabajo           := "INICIZA",
           SENSOR                   := DB2.DBX 4.0,
           PLANCHAS                 := "PLANCHAS");
      FP    "INICIZA";
NETWORK
TITLE =
      A     "X23";
      CALL  "CIZALLADO" , DB 6 (
           bit_de_trabajo           := "INICIZA",
           SENSOR                   := DB2.DBX 4.0,
           PLANCHAS                 := "PLANCHAS");
      FP    "INICIZA";
NETWORK
TITLE =
      A     "X23";
      CALL  "CIZALLADO" , DB 6 (
           bit_de_trabajo           := "INICIZA",
           SENSOR                   := DB3.DBX 4.0,
           PLANCHAS                 := "PLANCHAS");
      FP    "INICIZA";
NETWORK
TITLE =
      A     "X24";
      CALL  "CIZALLADO" , DB 6 (
           bit_de_trabajo           := "INICIZA",
           SENSOR                   := DB4.DBX 4.0,
           PLANCHAS                 := "PLANCHAS");
      FP    "INICIZA";
END_ORGANIZATION_BLOCK

ORGANIZATION_BLOCK "OB100"	// OB 100
TITLE = "Complete Restart"
VERSION : 0.1
VAR_TEMP
  OB100_EV_CLASS : BYTE ;	//16#13, Event class 1, Entering event state, Event logged in diagnostic buffer
  OB100_STRTUP : BYTE ;	//16#81/82/83/84 Method of startup
  OB100_PRIORITY : BYTE ;	//Priority of OB Execution
  OB100_OB_NUMBR : BYTE ;	//100 (Organization block 100, OB100)
  OB100_RESERVED_1 : BYTE ;	//Reserved for system
  OB100_RESERVED_2 : BYTE ;	//Reserved for system
  OB100_STOP : WORD ;	//Event that caused CPU to stop (16#4xxx)
  OB100_STRT_INFO : DWORD ;	//Information on how system started
  OB100_DATE_TIME : DATE_AND_TIME ;	//Date and time OB100 started
END_VAR
BEGIN
NETWORK
TITLE =
      SET;
      S     "X0";
      R     "X1";
      R     "X2";
      R     "X3";
      R     "X4";
      R     "X5";
      R     "X6";
      R     "X7";
      R     "X8";
      R     "X10";
      R     "X11";
      R     "X20";
      R     "X21";
      R     "X22";
      R     "X23";
      R     "X24";
      R     "X25";
      S     "X30";
      S     "X60";
      R     "X61";
      R     "X62";
      R     "X31";
      R     "X32";
      R     "X33";
      R     "X34";
      R     "X35";
      S     "X40";
      R     "X41";
      R     "X42";
      R     "X43";
      R     "X44";
      S     "X50";
      R     "X51";
      R     "X52";
      S     "X100";
      R     "X101";
      S     "X110";
      R     "X111";
      R     "X53";
      S     "X120";
      R     "ENDCOUNT";
      R     "X123";
      R     "X124";
      R     "X122";
      R     "X121";
      R     "X54";
      R     "STBYDESBOB";
      R     "INIDESBOB";
      R     "INICIZA";
      R     "SARTEN";
      R     "CACEROLA";
      R     "WOK";
      R     "PAELLERA";
      R     "CORTADO";
END_ORGANIZATION_BLOCK
